// Mitsubishi GX Works2 project: 서보모터펄스제어   PLC: Q02/Q02H

PROGRAM MAIN
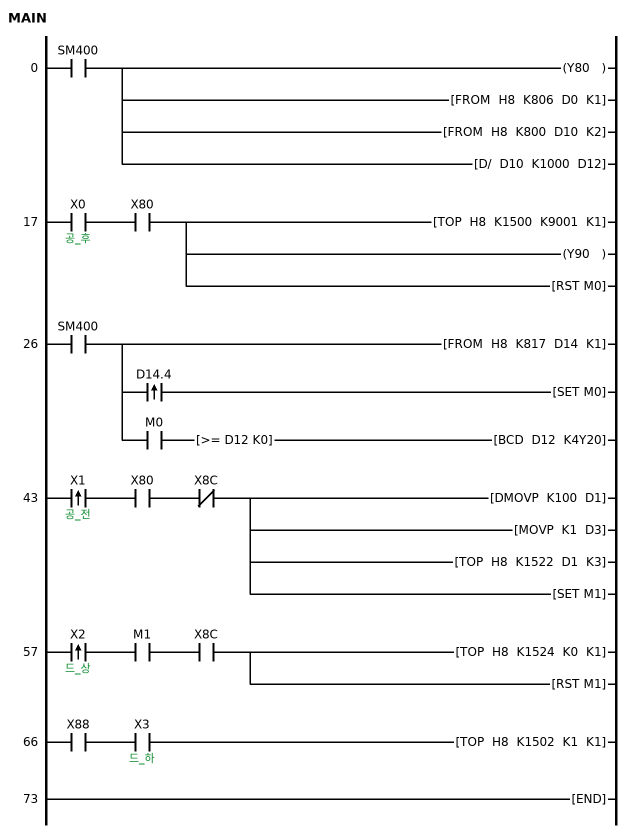
0     LD      SM400
      OUT     Y80
      FROM    H8 K806 D0 K1
      FROM    H8 K800 D10 K2
      D/      D10 K1000 D12
17    LD      X0  ; 공_후
      AND     X80
      TOP     H8 K1500 K9001 K1
      OUT     Y90
      RST     M0
26    LD      SM400
      FROM    H8 K817 D14 K1
      MPS
      ANDP    D14.4
      SET     M0
      MPP
      AND     M0
      AND>=   D12 K0
      BCD     D12 K4Y20  ; 공급_전
43    LDP     X1  ; 공_전
      AND     X80
      ANI     X8C
      DMOVP   K100 D1
      MOVP    K1 D3
      TOP     H8 K1522 D1 K3
      SET     M1
57    LDP     X2  ; 드_상
      AND     M1
      AND     X8C
      TOP     H8 K1524 K0 K1
      RST     M1
66    LD      X88
      AND     X3  ; 드_하
      TOP     H8 K1502 K1 K1
73    END
END_PROGRAM

// device comments not shown above
X4  ; 송_후
X5  ; 송_전
X6  ; 배_후
X7  ; 배_전
X8  ; 스_상
X9  ; 스_하
X0A  ; 흡_후
X0B  ; 흡_전
X0C  ; 창_후
X0D  ; 창_전
X0E  ; 용량형
X0F  ; 유도형
X1E  ; 스톱검출
X1F  ; 메거진
Y21  ; 공급_후
Y22  ; 드릴_하
Y23  ; 송출_전
Y24  ; 송출_후
Y25  ; 배출_전
Y26  ; 배출_후
Y27  ; 스_하
Y28  ; 흡_전
Y29  ; 흡_후
Y2A  ; 패드
Y2B  ; 창전
Y2C  ; 창후
Y2D  ; 드릴
Y2F  ; 컨베
